(* CODESYS project librarymotion.library
   Title: lcls-twincat-motion
   Version: 0.3.0
   Placeholder: lcls-twincat-motion
   Company: SLAC

Project tree, tasks and I/O mapping:
  libraries: Tc2_EtherCAT, * (Beckhoff Automation GmbH); Tc2_MC2, * (Beckhoff Automation GmbH); Tc2_Standard, * (Beckhoff Automation GmbH); Tc2_System, * (Beckhoff Automation GmbH); Tc2_Utilities, * (Beckhoff Automation GmbH); Tc3_Module, * (Beckhoff Automation GmbH)
  DUTs/
    data type DUT_MotionStage
    data type DUT_PositionState
    data type EL5042_Status
    data type ENUM_EpicsHomeCmd
    data type ENUM_EpicsMotorCmd
    data type ENUM_StageBrakeMode
    data type ENUM_StageEnableMode
    data type ST_RenishawAbsEnc
  POUs/
    Motion/
      Gantry/
        function block FB_GantryAutoCoupling [ST]
        function block FB_GantryDiffVirtualLimitSwitch [ST]
      function block FB_MotionStage [ST]
      function block FB_SetEnables [ST]
      function block FB_StatePTPMove [ST]
    MotorTesting/
      function block FB_MicroStepCountTest [ST]
  tc_mca_std_lib/
    DUTs/
    GVLs/
    POUs/
      ChangeConfig/
      ErrorHandling/
      Hardware/
        EtherCAT_Terminals/
          Analog_Inputs/
          Digital_Inputs/
          Digital_Outputs/
            External_Types/
          Measuring_Terminals/
          Motion/
          System/
        Other/
      Motion/
        Homing/
  UnitTests/
    program Interactive [ST]
  Version/
    global variables Global_Version
*)

// DUTs/DUT_MotionStage
TYPE DUT_MotionStage :
STRUCT
	(* Hardware *)
	
	// PLC Axis Reference
	Axis: AXIS_REF;
	// NC Forward Limit Switch: TRUE if ok to move
	{attribute 'pytmc': '
		pv: PLC:bLimitForwardEnable
		io: i
	'}
	bLimitForwardEnable AT %I*: BOOL;
	// NC Backward Limit Switch: TRUE if ok to move
	{attribute 'pytmc': '
		pv: PLC:bLimitBackwardEnable
		io: i
	'}
	bLimitBackwardEnable AT %I*: BOOL;
	// NO Home Switch: TRUE if at home
	{attribute 'pytmc': '
		pv: PLC:bHome
		io: i
	'}
	bHome AT %I*: BOOL;
	// NC Brake Output: TRUE to release brake
	{attribute 'pytmc': '
		pv: PLC:bBrakeRelease
		io: i
	'}
	bBrakeRelease AT %Q*: BOOL;
	// NC STO Input: TRUE if ok to move
	{attribute 'pytmc': '
		pv: PLC:bHardwareEnable
		io: i
	'}
	bHardwareEnable AT %I*: BOOL;

	(* Psuedo-hardware *)
	
	// Forward enable EPS summary
	{attribute 'pytmc': '
		pv: PLC:bAllForwardEnable
		io: i
	'}
	bAllForwardEnable: BOOL:=FALSE;
	// Backward enable EPS summary
	{attribute 'pytmc': '
		pv: PLC:bAllBackwardEnable
		io: i
	'}
	bAllBackwardEnable: BOOL:=FALSE; 
	// Enable EPS summary encapsulating emergency stop button and any additional motion preventive hardware
	{attribute 'pytmc': '
		pv: PLC:bAllEnable
		io: i
	'}
	bAllEnable: BOOL:=FALSE;
	// Forward virtual gantry limit switch
	{attribute 'pytmc': '
		pv: PLC:bGantryForwardEnable
		io: i
	'}
	bGantryForwardEnable: BOOL:=FALSE;
	// Backward virtual gantry limit switch
	{attribute 'pytmc': '
		pv: PLC:bGantryBackwardEnable
		io: i
	'}
	bGantryBackwardEnable: BOOL:=FALSE;
	
	(* Settings *)
	// Change to FALSE if MC_POWER is somewhere else in the project
	{attribute 'pytmc': '
		pv: PLC:bPowerSelf
		io: i
	'}
	bPowerSelf: BOOL:=TRUE;
	// Determines when we automatically enable the motor
	{attribute 'pytmc': '
		pv: PLC:nEnableMode
		io: i
	'}
	nEnableMode: INT:=ENUM_StageEnableMode.STAGE_ENABLE_MOTION;
	// Determines when we automatically disengage the brake
	{attribute 'pytmc': '
		pv: PLC:nBrakeMode
		io: i
	'}
	nBrakeMode: INT:=ENUM_StageBrakeMode.STAGE_BRAKE_DISABLED;
	// Determines our encoder homing strategy
	{attribute 'pytmc': '
		pv: PLC:nHomingMode
		io: i
	'}
	nHomingMode: INT:=ENUM_EpicsHomeCmd.EPICS_MOTOR_HOME_NONE;
	// Set true to activate gantry EPS
	{attribute 'pytmc': '
		pv: PLC:bGantryAxis
		io: i
	'}
	bGantryAxis: BOOL:=FALSE;
	// Set to gantry difference tolerance
	{attribute 'pytmc': '
		pv: PLC:nGantryTol
		io: i
	'}
	nGantryTol: LINT:=0;
	// Encoder count at which this axis is aligned with other axis
	{attribute 'pytmc': '
		pv: PLC:nEncRef
		io: i
	'}
	nEncRef: ULINT:=0;
	
	(* Commands *)
	// Used internally to request enables
	{attribute 'pytmc': '
		pv: PLC:bEnable
		io: io
	'}
	bEnable: BOOL;
	// Used internally to reset errors and other state
	{attribute 'pytmc': '
		pv: PLC:bReset
		io: io
	'}
	bReset: BOOL;
	// Used internally and by the IOC to start or stop a move
	{attribute 'pytmc': '
		pv: PLC:bExecute
		io: io
	'}
	bExecute: BOOL;
	
	(* Command Args *)
	// Used internally and by the IOC to pick what kind of move to do
	{attribute 'pytmc': '
		pv: PLC:nCommand
		io: io
	'}
	nCommand: INT;
	// Used internally and by the IOC to pass additional data to some commands
	{attribute 'pytmc': '
		pv: PLC:nCmdData
		io: io
	'}
	nCmdData: INT;
	// Used internally and by the IOC to pick a destination for the move
	{attribute 'pytmc': '
		pv: PLC:fPosition
		io: io
	'}
	fPosition: LREAL;
	// Used internally and by the IOC to pick a move velocity
	{attribute 'pytmc': '
		pv: PLC:fVelocity
		io: io
	'}
	fVelocity: LREAL;
	// Used internally and by the IOC to pick a move acceleration
	{attribute 'pytmc': '
		pv: PLC:fAcceleration
		io: io
	'}
	fAcceleration: LREAL;
	// Used internally and by the IOC to pick a move deceleration
	{attribute 'pytmc': '
		pv: PLC:fDeceleration
		io: io
	'}
	fDeceleration: LREAL;
	// Used internally and by the IOC to pick a home position
	{attribute 'pytmc': '
		pv: PLC:fHomePosition
		io: io
	'}
	fHomePosition: LREAL;
	
	(* Info *)
	// Unique ID assigned to each axis in the NC
	{attribute 'pytmc': '
		pv: PLC:nMotionAxisID
		io: i
	'}
	nMotionAxisID: UDINT:=0;
	
	(* Returns *)
	// TRUE if done enabling
	{attribute 'pytmc': '
		pv: PLC:bEnableDone
		io: i
	'}
	bEnableDone: BOOL;
	// TRUE if in the middle of a command
	{attribute 'pytmc': '
		pv: PLC:bBusy
		io: i
	'}
	bBusy: BOOL;
	// TRUE if we've done a command and it has finished
	{attribute 'pytmc': '
		pv: PLC:bDone
		io: i
	'}
	bDone: BOOL;
	// TRUE if we're in an error state
	{attribute 'pytmc': '
		pv: PLC:bError
		io: i
	'}
	bError: BOOL;
	// Message to identify the error state
	{attribute 'pytmc': '
		pv: PLC:sErrorMessage
		io: i
	'}
	sErrorMessage: STRING;
	// Misc axis status information for the IOC
	stAxisStatus: DUT_AxisStatus_v0_01;
END_STRUCT
END_TYPE

// DUTs/DUT_PositionState
TYPE DUT_PositionState :
// Include io: input on things that should never be mutable in EPICS.
// Omit io on things that may or may not need to be mutable, allow engineer to decide in their pragma.
// Currently: some installations would want position and delta to be mutable.
STRUCT
	{attribute 'pytmc' := '
		pv: NAME
		io: input
	'}
	sName: STRING;

	{attribute 'pytmc' := '
		pv: SETPOINT
		io: io
	'}
	fPosition: LREAL;
	
	{attribute 'pytmc' := '
		pv: DELTA
		io: io
	'}
	fDelta: LREAL;
	
	{attribute 'pytmc' := '
		pv: VELO
		io: io
	'}
	fVelocity: LREAL;
	
	{attribute 'pytmc' := '
		pv: ACCL
		io: io
	'}
	fAccel: LREAL;
	
	{attribute 'pytmc' := '
		pv: DCCL
		io: io
	'}
	fDecel: LREAL;
END_STRUCT
END_TYPE

// DUTs/EL5042_Status
TYPE EL5042_Status :
STRUCT
END_STRUCT
END_TYPE

// DUTs/ENUM_EpicsHomeCmd
{attribute 'qualified_only'}
{attribute 'strict'}
TYPE ENUM_EpicsHomeCmd :
(
	EPICS_MOTOR_HOME_LLS := 1, // Low limit switch
	EPICS_MOTOR_HOME_HLS := 2, // High limit switch
	EPICS_MOTOR_HOME_LHS := 3, // Home switch via low switch
	EPICS_MOTOR_HOME_HHS := 4, // Home switch via high switch
	EPICS_MOTOR_HOME_ABS := 15, // Set here to be fHomePosition
	EPICS_MOTOR_HOME_NONE := -1 // Do not home, ever
);
END_TYPE

// DUTs/ENUM_EpicsMotorCmd
{attribute 'qualified_only'}
{attribute 'strict'}
TYPE ENUM_EpicsMotorCmd :
(
	EPICS_MOTOR_JOG := 0,
	EPICS_MOTOR_MOVE_VEL := 1,
	EPICS_MOTOR_MOVE_REL := 2,
	EPICS_MOTOR_MOVE_ABS := 3,
	EPICS_MOTOR_MOVE_MOD := 4,
	EPICS_MOTOR_HOME := 10,
	EPICS_MOTOR_GEAR := 30
);
END_TYPE

// DUTs/ENUM_StageBrakeMode
{attribute 'qualified_only'}
{attribute 'strict'}
TYPE ENUM_StageBrakeMode :
(
	STAGE_BRAKE_DISABLED,
	STAGE_BRAKE_STANDSTILL
);
END_TYPE

// DUTs/ENUM_StageEnableMode
{attribute 'qualified_only'}
{attribute 'strict'}
TYPE ENUM_StageEnableMode :
(
	STAGE_ENABLE_ALWAYS, // Always set bEnable to TRUE
	STAGE_ENABLE_NEVER,  // Only change bEnable on errors
	STAGE_ENABLE_MOTION  // Enable before motion, disable after motion
);
END_TYPE

// DUTs/ST_RenishawAbsEnc
// Renishaw BiSS-C absolute encoder used with an EL5042 
TYPE ST_RenishawAbsEnc :
STRUCT
	Count AT %I*: ULINT; // Connect to encoder "Position" input
	Status: EL5042_Status; // Status struct placeholder
	Ref: ULINT; // Encoder zero position (useful for aligned position with gantries)
END_STRUCT
END_TYPE

// Version/Global_Version
{attribute 'TcGenerated'}
// This function has been automatically generated from the project information.
VAR_GLOBAL CONSTANT
	{attribute 'const_non_replaced'}
	{attribute 'linkalways'
	stLibVersion_lcls-twincat-motion : ST_LibVersion := (iMajor := 0, iMinor := 3, iBuild := 0, iRevision := 0, sVersion := '0.3.0');
END_VAR

// POUs/Motion/Gantry/FB_GantryAutoCoupling
FUNCTION_BLOCK FB_GantryAutoCoupling
VAR_INPUT
	nGantryTol : LINT;
END_VAR
VAR_OUTPUT
	bGantryAlreadyCoupled : BOOL;
END_VAR
VAR_IN_OUT
	Master : DUT_MotionStage;
	MasterEnc : ST_RenishawAbsEnc;
	Slave : DUT_MotionStage;
	SlaveEnc : ST_RenishawAbsEnc;
	bExecuteCouple : BOOL;
	bExecuteDecouple : BOOL;
END_VAR
VAR
	gantry_diff_limit : FB_GantryDiffVirtualLimitSwitch;
	couple : MC_GEARIN;
	decouple : MC_GEAROUT;
	bInitComplete : BOOL;
	fbSetEnables : FB_SetEnables;
END_VAR

// Designate Master and SLave Axes
Master.bGantryAxis := TRUE;
Slave.bGantryAxis := TRUE;

Master.nGantryTol := nGantryTol;
Slave.nGantryTol := Master.nGantryTol;

// Activate Gantry Virtual Limit Switch
gantry_diff_limit(Penc:=MasterEnc, SEnc:=SlaveEnc, GantDiffTol:=Master.nGantryTol,
				  PLimFwd=>Master.bGantryForwardEnable, PLimBwd=>Master.bGantryBackwardEnable,
				  SLimFwd=>Slave.bGantryForwardEnable, SLimBwd=>Slave.bGantryBackwardEnable);

// Coupling Status Bit
bGantryAlreadyCoupled := Master.Axis.NcToPlc.CoupleState=1 AND Slave.Axis.NcToPlc.CoupleState=3;

fbSetEnables(stMotionStage:=Master);
fbSetEnables(stMotionStage:=Slave);

IF bGantryAlreadyCoupled THEN
	Master.bGantryForwardEnable := Master.bGantryForwardEnable AND Slave.bAllForwardEnable;
	Slave.bGantryForwardEnable := Master.bAllForwardEnable AND Slave.bGantryForwardEnable;
	
	Master.bGantryBackwardEnable := Master.bGantryBackwardEnable AND Slave.bAllBackwardEnable;
	Slave.bGantryBackwardEnable := Master.bAllBackwardEnable AND Slave.bGantryBackwardEnable;
END_IF


// Coupling states
// Auto-coupling at init and auto-reset of coupling boolean
bExecuteCouple S= NOT bInitComplete;

bExecuteCouple R= couple.Busy OR bGantryAlreadyCoupled;
couple(Master:=Master.Axis, Slave:=Slave.Axis, Execute:=bExecuteCouple);

bInitComplete S= bGantryAlreadyCoupled;

// Decoupling with auto-reset of coupling boolean
bExecuteDecouple R= decouple.Busy OR NOT bGantryAlreadyCoupled;
decouple(Slave:=Slave.Axis, Execute:=bExecuteDecouple);

END_FUNCTION_BLOCK

// POUs/Motion/Gantry/FB_GantryDiffVirtualLimitSwitch
FUNCTION_BLOCK FB_GantryDiffVirtualLimitSwitch
VAR_INPUT
	PEnc: ST_RenishawAbsEnc; // Primary axis encoder (usually the upstream one)
	SEnc: ST_RenishawAbsEnc; // Secondary axis encoder (couples to the primary)
	
	GantDiffTol: LINT;		// Gantry differenace tolerance in encoder counts
END_VAR
VAR_OUTPUT
	PLimFwd: BOOL; // Primary axis forward direction enable
	PLimBwd: BOOL; // Primary axis reverse direction enable
	SLimFwd: BOOL; // Secondary axis forward direction enable
	SLimBwd: BOOL; // Secondary axis reverse direction enable
END_VAR
VAR
	GantryDiff: LINT;
END_VAR

(* Gantry Difference Virtual Limit Switch
A. Wallace 2017-2-15

Determines which direction is disabled due to it increasing the gantry difference.
Refer to the ESD for actual conventions.

A positive gantry error refers to a CCW clocked assembly:
eg. for X
X1 upstream, X2 downstream. Primary axis is always upstream.
Gantry difference > 0 when
X2>X1
Therefore
X2 positive direction disabled
X1 negative direction disabled

Call before FB_MotionStage fb calls for the gantry axes.
*)

GantryDiff := ( ULINT_TO_LINT(PEnc.Count) - ULINT_TO_LINT(PEnc.Ref) ) - ( ULINT_TO_LINT(SEnc.Count) - ULINT_TO_LINT(SEnc.Ref) );

IF ABS(GantryDiff) > GantDiffTol THEN
	IF GantryDiff < 0  THEN
		PLimBwd := FALSE;
		SLimFwd := FALSE;
	ELSE	
		PLimBwd := TRUE;
		SLimFwd := TRUE;
	END_IF
	IF GantryDiff > 0 THEN
		PLimFwd := FALSE;
		SLimBwd := FALSE;
	ELSE
		PLimFwd := TRUE;
		SLimBwd := TRUE;
	END_IF
ELSE
	//If there is no fault, all directions are enabled
	PLimFwd := TRUE;
	PLimBwd := TRUE;
	SLimFwd := TRUE;
	SLimBwd := TRUE;
END_IF

END_FUNCTION_BLOCK

// POUs/Motion/FB_MotionStage
FUNCTION_BLOCK FB_MotionStage
VAR_IN_OUT
	stMotionStage: DUT_MotionStage;
END_VAR
VAR
	fbDriveVirtual: FB_DriveVirtual;
	bExecute: BOOL;
	bFwdHit: BOOL;
	bBwdHit: BOOL;
	fbExecFallingEdge: F_TRIG;
	fbSetEnables: FB_SetEnables;
END_VAR

// Start with an accurate status
stMotionStage.Axis.ReadStatus();

// Handle auto-enable timing
CASE stMotionStage.nEnableMode OF
	ENUM_StageEnableMode.STAGE_ENABLE_ALWAYS:
		stMotionStage.bEnable := TRUE;
		bExecute := stMotionStage.bExecute;
	ENUM_StageEnableMode.STAGE_ENABLE_NEVER:
		bExecute := stMotionStage.bExecute;
	ENUM_StageEnableMode.STAGE_ENABLE_MOTION:
		IF stMotionStage.bExecute THEN
			stMotionStage.bEnable := TRUE;
		END_IF
		bExecute := stMotionStage.bExecute AND stMotionStage.bEnableDone;
END_CASE

// Automatically fill the correct nCmdData for homing
IF stMotionStage.nCommand = ENUM_EpicsMotorCmd.EPICS_MOTOR_HOME THEN
	stMotionStage.nCmdData := stMotionStage.nHomingMode;
END_IF

fbSetEnables(stMotionStage:=stMotionStage);

// Handle standard commands using ESS's FB
fbDriveVirtual(En:=TRUE,
	bEnable:=stMotionStage.bAllEnable,
	bReset:=stMotionStage.bReset,
	bExecute:=bExecute,
	nCommand:=INT_TO_UINT(stMotionStage.nCommand),
	nCmdData:=INT_TO_UINT(stMotionStage.nCmdData),
	fVelocity:=stMotionStage.fVelocity,
	fPosition:=stMotionStage.fPosition,
	fAcceleration:=stMotionStage.fAcceleration,
	fDeceleration:=stMotionStage.fDeceleration,
	bLimitFwd:=stMotionStage.bAllForwardEnable,
	bLimitBwd:=stMotionStage.bAllBackwardEnable,
	bHomeSensor:=stMotionStage.bHome,
	fHomePosition:=stMotionStage.fHomePosition,
	bPowerSelf:=stMotionStage.bPowerSelf,
	nMotionAxisID=>stMotionStage.nMotionAxisID,
	bError=>stMotionStage.bError,
	sErrorMessage=>stMotionStage.sErrorMessage,
	Axis:=stMotionStage.Axis);

IF fbDriveVirtual.bBusy THEN
	stMotionStage.bBusy := TRUE;
	stMotionStage.bDone := FALSE;
END_IF

IF stMotionStage.bError THEN
	stMotionStage.bBusy := FALSE;
	stMotionStage.bDone := FALSE;
	stMotionStage.bEnable := FALSE;
END_IF

// Check the limits and cancel execution if appropriate. Without this block we have infinite error spam
bFwdHit := stMotionStage.Axis.Status.PositiveDirection AND NOT stMotionStage.bAllForwardEnable;
bBwdHit := stMotionStage.Axis.Status.NegativeDirection AND NOT stMotionStage.bAllBackwardEnable;
IF bFwdHit OR bBwdHit THEN
	stMotionStage.bExecute := FALSE;
END_IF

// Mark done if settled or if unexpected stop, then reset the FB if there is no error
fbExecFallingEdge(CLK:=stMotionStage.bExecute);
IF (stMotionStage.Axis.Status.InTargetPosition AND NOT fbDriveVirtual.bBusy) OR fbExecFallingEdge.Q THEN
	IF NOT stMotionStage.bDone THEN
		stMotionStage.bDone := TRUE;
		stMotionStage.bBusy := FALSE;
		IF NOT stMotionStage.Axis.Status.Error THEN
			bExecute := FALSE;
			stMotionStage.bExecute := FALSE;
		END_IF
	END_IF
END_IF
IF stMotionStage.nEnableMode = ENUM_StageEnableMode.STAGE_ENABLE_MOTION AND NOT bExecute THEN
	IF stMotionStage.Axis.Status.MotionState = MC_AXISSTATE_STANDSTILL THEN
		stMotionStage.bEnable := FALSE;
	END_IF
END_IF

// Get a definitive bEnabled reading
CASE stMotionStage.Axis.Status.MotionState OF
	// We are not enabled if there is an issue
	MC_AXISSTATE_UNDEFINED, MC_AXISSTATE_DISABLED, MC_AXISSTATE_ERRORSTOP:
		stMotionStage.bEnableDone := FALSE;
	ELSE
		stMotionStage.bEnableDone := TRUE;
END_CASE

// Handle the brake. TRUE means brake disabled.
CASE stMotionStage.nBrakeMode OF
	ENUM_StageBrakeMode.STAGE_BRAKE_DISABLED:
		stMotionStage.bBrakeRelease := stMotionStage.bEnableDone AND stMotionStage.bExecute;
	ENUM_StageBrakeMode.STAGE_BRAKE_STANDSTILL:
		IF stMotionStage.Axis.Status.MotionState = MC_AXISSTATE_STANDSTILL THEN
			stMotionStage.bBrakeRelease := FALSE;
		ELSE
			stMotionStage.bBrakeRelease := TRUE;
		END_IF
END_CASE
CASE stMotionStage.Axis.Status.MotionState OF
	MC_AXISSTATE_UNDEFINED, MC_AXISSTATE_ERRORSTOP:
		stMotionStage.bBrakeRelease := FALSE;
END_CASE

// Sync the epics status struct
stMotionStage.stAxisStatus := fbDriveVirtual.stAxisStatus;
stMotionStage.stAxisStatus.bEnabled := stMotionStage.bEnableDone;

// Reset everything when bReset is flagged
IF stMotionStage.bReset THEN
	stMotionStage.bEnable := FALSE;
	stMotionStage.bReset := FALSE;
	stMotionStage.bExecute := FALSE;
	bExecute := FALSE;
END_IF

// Ignore homing if we have the setting for it
// e.g. for pre-calibrated absolute encoders
IF stMotionStage.nHomingMode = ENUM_EpicsHomeCmd.EPICS_MOTOR_HOME_NONE THEN
	stMotionStage.stAxisStatus.bHomed := TRUE;
END_IF

END_FUNCTION_BLOCK

// POUs/Motion/FB_SetEnables
FUNCTION_BLOCK FB_SetEnables
VAR_IN_OUT
	stMotionStage: DUT_MotionStage;
END_VAR

stMotionStage.bAllForwardEnable := stMotionStage.bLimitForwardEnable AND (stMotionStage.bGantryForwardEnable OR NOT stMotionStage.bGantryAxis);
stMotionStage.bAllBackwardEnable := stMotionStage.bLimitBackwardEnable AND (stMotionStage.bGantryBackwardEnable OR NOT stMotionStage.bGantryAxis);

stMotionStage.bAllEnable := stMotionStage.bEnable AND stMotionStage.bHardwareEnable;

END_FUNCTION_BLOCK

// POUs/Motion/FB_StatePTPMove
FUNCTION_BLOCK FB_StatePTPMove
// For your pytmc pragma on this block, specify io accordingly:
// 1. use input or i if you want the set position to be immutable
// 2. use io if you want to set position to be mutable from epics
VAR_INPUT
	{attribute 'pytmc' := '
		pv:
	'}
	stPositionState: DUT_PositionState;
	
	{attribute 'pytmc' := '
		pv: GO
		io: io
		field: ZNAM False
		field: ONAM True
	'}
	bExecute: BOOL;
	
	{attribute 'pytmc' := '
		pv: MOVE_OK
		io: input
		field: ZNAM False
		field: ONAM True
	'}
	bMoveOk: BOOL;
END_VAR
VAR_IN_OUT
	stMotionStage: DUT_MotionStage;
END_VAR
VAR_OUTPUT
	{attribute 'pytmc' := '
		pv: AT_STATE
		io: input
		field: ZNAM False
		field: ONAM True
	'}
	bAtState: BOOL;
	
	{attribute 'pytmc' := '
		pv: DMOV
		io: input
		field: ZNAM False
		field: ONAM True
	'}
	bDone: BOOL;
	
	{attribute 'pytmc' := '
		pv: BUSY
		io: input
		field: ZNAM False
		field: ONAM True
	'}
	bBusy: BOOL;
	
	{attribute 'pytmc' := '
		pv: ERR
		io: input
		field: ZNAM False
		field: ONAM True
	'}
	bError: BOOL;
	
	{attribute 'pytmc' := '
		pv: ERRMSG
		io: input
	'}
	sError: STRING;
END_VAR
VAR
	bExecTrig: R_TRIG;
	bExecEnd: F_TRIG;
	fActPosition: LREAL;
	fLowPos: LREAL;
	fHighPos: LREAL;
END_VAR

bExecTrig(CLK:=bExecute);
IF bExecTrig.Q AND bMoveOk THEN
	IF NOT stMotionStage.bBusy AND NOT stMotionStage.bError THEN
		stMotionStage.bExecute := TRUE;
		stMotionStage.nCommand := ENUM_EpicsMotorCmd.EPICS_MOTOR_MOVE_ABS;
		stMotionStage.fPosition := stPositionState.fPosition;
		stMotionStage.fVelocity := stPositionState.fVelocity;
		stMotionStage.fAcceleration := stPositionState.fAccel;
		stMotionStage.fDeceleration := stPositionState.fDecel;
		bDone := FALSE;
		bBusy := TRUE;
	END_IF
END_IF
bError := stMotionStage.bError;
sError := stMotionStage.sErrorMessage;

fActPosition := stMotionStage.stAxisStatus.fActPosition;
fLowPos := stPositionState.fPosition - stPositionState.fDelta;
fHighPos := stPositionState.fPosition + stPositionState.fDelta;
IF (fLowPos < fActPosition) AND (fHighPos > fActPosition) THEN
	bAtState := TRUE;
	IF NOT stMotionStage.bBusy THEN
		bDone := TRUE;
		bBusy := FALSE;
		bExecute := FALSE;
	END_IF
ELSE
	bAtState := FALSE;
END_IF

bExecEnd(CLK:=bExecute);
IF bExecEnd.Q AND bBusy THEN
	stMotionStage.bExecute := FALSE;
END_IF

IF NOT stMotionStage.bExecute OR NOT bExecute THEN
	bDone := TRUE;
	bBusy := FALSE;
	bExecute := FALSE;
END_IF

END_FUNCTION_BLOCK

// POUs/MotorTesting/FB_MicroStepCountTest
FUNCTION_BLOCK FB_MicroStepCountTest
VAR_INPUT
	bExecute: BOOL;
	fStepSize: LREAL;
	nSteps: UINT;
	fMicroStep: LREAL;
	fVelocity: LREAL;
	tSettleTime: TIME;
END_VAR
VAR_IN_OUT
	Axis: AXIS_REF;
END_VAR
VAR_OUTPUT
	nStepsCounted: UINT;
	nTheorySteps: UINT;
	fPercent: LREAL;
	fEstMicroSize: LREAL;
END_VAR
VAR
	fbMoveRel: MC_MoveRelative;
	fbSettleTimer: TON;
	bDoMove: BOOL;
	nStepCounter: UINT;
	
	arrPosBuffer: ARRAY [0..99] OF LREAL;
	fAvgPos: LREAL;
	nArrIndex: UINT;
	nLoopIndex: UINT;
	
	fStartPos: LREAL;
	fPrevPos: LREAL;
	fStepChange: LREAL;
	
	fStepSum: LREAL;
END_VAR

// Motion FB
fbMoveRel(Axis:=Axis,
	Execute:=bDoMove,
	Distance:=fStepSize,
	Velocity:=fVelocity);
	
// Settle time
fbSettleTimer(IN:=fbMoveRel.Done,
	PT:=tSettleTime);
	
// Re-enable the move for next cycle
bDoMove := bExecute AND nStepCounter < nSteps;

// Calculate rolling average
arrPosBuffer[nArrIndex] := Axis.NcToPlc.ActPos;
fAvgPos := 0;
FOR nLoopIndex := 0 TO 99 DO
	fAvgPos := fAvgPos + arrPosBuffer[nLoopIndex];
END_FOR;
fAvgPos := fAvgPos / 100;
nArrIndex := (nArrIndex + 1) MOD 100;

// Initialize starting variables
IF NOT bExecute THEN
	fStartPos := fAvgPos;
	fPrevPos := fAvgPos;
END_IF

// Check results
IF fbSettleTimer.Q THEN
	fStepChange := fAvgPos - fPrevPos;
	// Invert fStepChange if we were doing negative steps
	IF fStepSize < 0 THEN
		fStepChange := fStepChange * -1;
	END_IF
	IF fStepChange > fMicroStep * 0.5 THEN
		nStepsCounted := nStepsCounted + 1;
		fStepSum := fStepSum + fStepChange;
		fEstMicroSize := fStepSum / nStepsCounted;
	END_IF
	nTheorySteps := DINT_TO_UINT(TRUNC(ABS((fStartPos - fAvgPos) / fMicroStep)));
	IF nTheorySteps > 0 THEN
		fPercent := 100 * nStepsCounted / nTheorySteps;
	END_IF
	fPrevPos := fAvgPos;
	nStepCounter := nStepCounter + 1;
	// Reset the move block
	bDoMove := FALSE;
END_IF

END_FUNCTION_BLOCK

// UnitTests/Interactive
PROGRAM Interactive
VAR
	M1: DUT_MotionStage;
	fbMotionStage: FB_MotionStage;
	nCounter: UINT;
	
	stOut: DUT_PositionState;
	fbGoOut: FB_StatePTPMove;
	bOut: BOOL;
	bGoOut: BOOL;
	stIn: DUT_PositionState;
	fbGoIn: FB_StatePTPMove;
	bIn: BOOL;
	bGoIn: BOOL;
	stUnsafe: DUT_PositionState;
	fbGoBad: FB_StatePTPMove;
	bHCF: BOOL;
	bGoHCF: BOOL;
END_VAR

M1.bPowerSelf := TRUE;
M1.bLimitBackwardEnable := TRUE;
M1.bLimitForwardEnable := TRUE;
fbMotionStage(stMotionStage:=M1);
nCounter := nCounter + 1;

stOut.sName := 'Out';
stOut.fPosition := 100;
stOut.fDelta := 20;
stOut.fVelocity := 10;

stIn.sName := 'In';
stIn.fPosition := 0;
stIn.fDelta := 0.1;
stIn.fVelocity := 5;

stUnsafe.sName := 'HCF';
stUnsafe.fPosition := -999;
stUnsafe.fDelta := 6;
stUnsafe.fVelocity := 42;

fbGoOut(
	bExecute:=bGoOut,
	stMotionStage:=M1,
	stPositionState:=stOut,
	bMoveOk:=TRUE,
	bAtState=>bOut);
fbGoIn(
	bExecute:=bGoIn,
	stMotionStage:=M1,
	stPositionState:=stIn,
	bMoveOk:=TRUE,
	bAtState=>bIn);
fbGoBad(
	bExecute:=bGoHCF,
	stMotionStage:=M1,
	stPositionState:=stUnsafe,
	bAtState=>bHCF);

END_PROGRAM
